// TIA Portal project "0511_grua" (V20)

(* hardware
DEVICE "S7-1200 station_1"  S7-1200 Station
   slot 0: "Rack_0"  S7-1200 Rack  Rack  V1.0
   slot 1: "PLC_1"  CPU 1215C AC/DC/Rly  6ES7 215-1BG40-0XB0  V4.7
*)

// ===== PLC "PLC_1"  CPU 1215C AC/DC/Rly =====

VAR_GLOBAL   // PLC tag table "Default tag table"
   "Etapa 0" AT %M0.0 : Bool;
   "Etapa 1" AT %M0.1 : Bool;
   "Etapa 2" AT %M0.2 : Bool;
   "Etapa 3" AT %M0.3 : Bool;
   "Etapa 4" AT %M0.4 : Bool;
   "Etapa 5" AT %M0.5 : Bool;
   "Etapa 6" AT %M0.6 : Bool;
   "Etapa 7" AT %M0.7 : Bool;
   "S1" AT %I0.0 : Bool;
   "FC1" AT %I0.1 : Bool;
   "FC2" AT %I0.2 : Bool;
   "FC3" AT %I0.3 : Bool;
   "FC4" AT %I0.4 : Bool;
   "Subir Grua" AT %Q0.0 : Bool;
   "Bajar Grua" AT %Q0.1 : Bool;
   "Mover Derecha" AT %Q0.2 : Bool;
   "Mover Izquierda" AT %Q0.3 : Bool;
END_VAR

// folder: System blocks/Program resources

DATA_BLOCK "IEC_Timer_0_DB"   // DB1
{ S7_Optimized_Access := 'TRUE' }
AUTHOR : Simatic
FAMILY : IEC
NAME : IEC_TMR
VERSION : 1.0
// stored: InstanceOfName IEC_TIMER
"IEC_TIMER"
BEGIN
END_DATA_BLOCK

// folder: (top level)

ORGANIZATION_BLOCK "Main"   // OB1, LAD, ProgramCycle
TITLE = "Main Program Sweep (Cycle)"
{ S7_Optimized_Access := 'TRUE' }
VERSION : 0.1
   VAR_INPUT
      Initial_Call : Bool;   // Initial call of this OB
      Remanence : Bool;   // =True, if remanent data are available
   END_VAR
BEGIN

REGION Network 1: Etapa 0
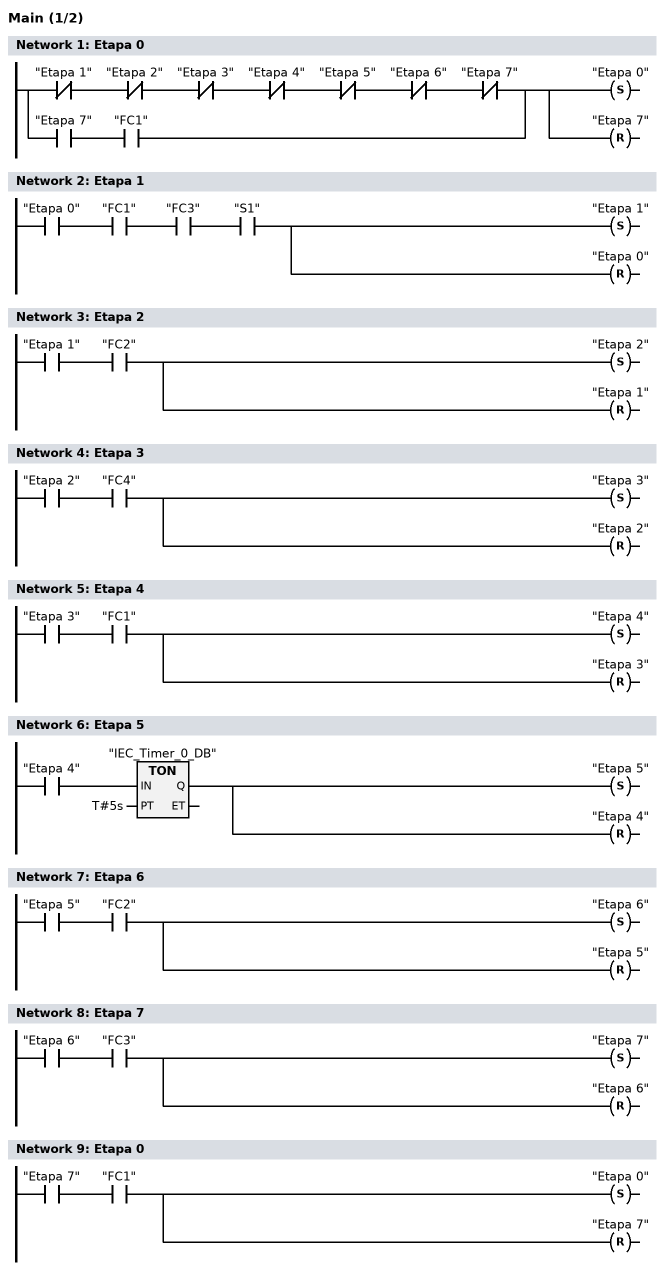
   RUNG wire#powerrail
      I_Contact( "Etapa 1" )
      I_Contact( "Etapa 2" )
      I_Contact( "Etapa 3" )
      I_Contact( "Etapa 4" )
      I_Contact( "Etapa 5" )
      I_Contact( "Etapa 6" )
      I_Contact( "Etapa 7" )
      wire#w1
      S_Coil( "Etapa 0" )
   END_RUNG
   RUNG wire#powerrail
      Contact( "Etapa 7" )
      Contact( "FC1" )
   END_RUNG wire#w1
   RUNG wire#w1
      R_Coil( "Etapa 7" )
   END_RUNG
   // the same network as SCL:
   IF (NOT "Etapa 1" AND NOT "Etapa 2" AND NOT "Etapa 3" AND NOT "Etapa 4" AND NOT "Etapa 5" AND NOT "Etapa 6" AND NOT "Etapa 7") OR ("Etapa 7" AND "FC1") THEN
       "Etapa 0" := TRUE;
       "Etapa 7" := FALSE;
   END_IF;
END_REGION

REGION Network 2: Etapa 1
   RUNG wire#powerrail
      Contact( "Etapa 0" )
      Contact( "FC1" )
      Contact( "FC3" )
      Contact( "S1" )
      wire#w1
      S_Coil( "Etapa 1" )
   END_RUNG
   RUNG wire#w1
      R_Coil( "Etapa 0" )
   END_RUNG
   // the same network as SCL:
   IF "Etapa 0" AND "FC1" AND "FC3" AND "S1" THEN
       "Etapa 1" := TRUE;
       "Etapa 0" := FALSE;
   END_IF;
END_REGION

REGION Network 3: Etapa 2
   RUNG wire#powerrail
      Contact( "Etapa 1" )
      Contact( "FC2" )
      wire#w1
      S_Coil( "Etapa 2" )
   END_RUNG
   RUNG wire#w1
      R_Coil( "Etapa 1" )
   END_RUNG
   // the same network as SCL:
   IF "Etapa 1" AND "FC2" THEN
       "Etapa 2" := TRUE;
       "Etapa 1" := FALSE;
   END_IF;
END_REGION

REGION Network 4: Etapa 3
   RUNG wire#powerrail
      Contact( "Etapa 2" )
      Contact( "FC4" )
      wire#w1
      S_Coil( "Etapa 3" )
   END_RUNG
   RUNG wire#w1
      R_Coil( "Etapa 2" )
   END_RUNG
   // the same network as SCL:
   IF "Etapa 2" AND "FC4" THEN
       "Etapa 3" := TRUE;
       "Etapa 2" := FALSE;
   END_IF;
END_REGION

REGION Network 5: Etapa 4
   RUNG wire#powerrail
      Contact( "Etapa 3" )
      Contact( "FC1" )
      wire#w1
      S_Coil( "Etapa 4" )
   END_RUNG
   RUNG wire#w1
      R_Coil( "Etapa 3" )
   END_RUNG
   // the same network as SCL:
   IF "Etapa 3" AND "FC1" THEN
       "Etapa 4" := TRUE;
       "Etapa 3" := FALSE;
   END_IF;
END_REGION

REGION Network 6: Etapa 5
   "IEC_Timer_0_DB".TON(IN := "Etapa 4", PT := T#5s);
   IF "IEC_Timer_0_DB".Q THEN
       "Etapa 5" := TRUE;
       "Etapa 4" := FALSE;
   END_IF;
END_REGION

REGION Network 7: Etapa 6
   RUNG wire#powerrail
      Contact( "Etapa 5" )
      Contact( "FC2" )
      wire#w1
      S_Coil( "Etapa 6" )
   END_RUNG
   RUNG wire#w1
      R_Coil( "Etapa 5" )
   END_RUNG
   // the same network as SCL:
   IF "Etapa 5" AND "FC2" THEN
       "Etapa 6" := TRUE;
       "Etapa 5" := FALSE;
   END_IF;
END_REGION

REGION Network 8: Etapa 7
   RUNG wire#powerrail
      Contact( "Etapa 6" )
      Contact( "FC3" )
      wire#w1
      S_Coil( "Etapa 7" )
   END_RUNG
   RUNG wire#w1
      R_Coil( "Etapa 6" )
   END_RUNG
   // the same network as SCL:
   IF "Etapa 6" AND "FC3" THEN
       "Etapa 7" := TRUE;
       "Etapa 6" := FALSE;
   END_IF;
END_REGION

REGION Network 9: Etapa 0
   RUNG wire#powerrail
      Contact( "Etapa 7" )
      Contact( "FC1" )
      wire#w1
      S_Coil( "Etapa 0" )
   END_RUNG
   RUNG wire#w1
      R_Coil( "Etapa 7" )
   END_RUNG
   // the same network as SCL:
   IF "Etapa 7" AND "FC1" THEN
       "Etapa 0" := TRUE;
       "Etapa 7" := FALSE;
   END_IF;
END_REGION

REGION Network 10: Subir Grua
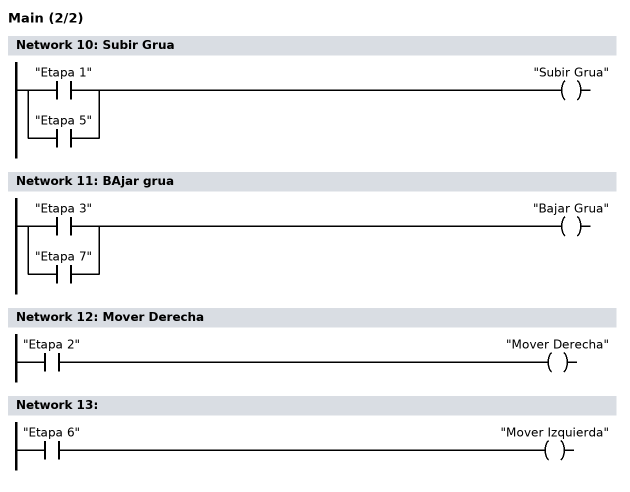
   RUNG wire#powerrail
      Contact( "Etapa 1" )
      wire#w1
      Coil( "Subir Grua" )
   END_RUNG
   RUNG wire#powerrail
      Contact( "Etapa 5" )
   END_RUNG wire#w1
   // the same network as SCL:
   "Subir Grua" := "Etapa 1" OR "Etapa 5";
END_REGION

REGION Network 11: BAjar grua
   RUNG wire#powerrail
      Contact( "Etapa 3" )
      wire#w1
      Coil( "Bajar Grua" )
   END_RUNG
   RUNG wire#powerrail
      Contact( "Etapa 7" )
   END_RUNG wire#w1
   // the same network as SCL:
   "Bajar Grua" := "Etapa 3" OR "Etapa 7";
END_REGION

REGION Network 12: Mover Derecha
   RUNG wire#powerrail
      Contact( "Etapa 2" )
      Coil( "Mover Derecha" )
   END_RUNG
   // the same network as SCL:
   "Mover Derecha" := "Etapa 2";
END_REGION

REGION Network 13
   RUNG wire#powerrail
      Contact( "Etapa 6" )
      Coil( "Mover Izquierda" )
   END_RUNG
   // the same network as SCL:
   "Mover Izquierda" := "Etapa 6";
END_REGION
END_ORGANIZATION_BLOCK